FUNCTION_BLOCK TFallingEdge
VAR
    F_TRIG1 : F_TRIG;
END_VAR

PROPERTY EdgeDetected : BOOL
GET
EdgeDetected := F_TRIG1.Q;
END_GET
END_PROPERTY

METHOD Test : BOOL
VAR_INPUT
    Value : BOOL;
END_VAR
F_TRIG1(CLK := Value);
Test := F_TRIG1.Q;
END_METHOD

END_FUNCTION_BLOCK

(* stored: Version 1.1.0.1, ProductVersion 3.1.4024.3
   POU TFallingEdge: Id {0a565260-f94b-034b-35fb-51ec95acf4da}, SpecialFunc None
   Property EdgeDetected: Id {8a7f01d2-2231-0532-02d7-e8b5bde55955}
   Get Get: Id {b2ae2c08-c211-0afc-1096-2bc7a2591a0a}
   Method Test: Id {6e01adbb-ead7-0505-0d79-1e7ea44ce992} *)
